FUNCTION F_ITC_SendRTR : BOOL
(**************************************************************************************
 * 	Application		:	BoxControl Framework
 *	Revision		:	$Revision: 404529 $
 *	Revision date	:	$Date: 2018-04-23 08:21:38 +0200 (Mo., 23 Apr 2018) $
 *	Last changed by	:	$Author: b7bolm $
 *	URL				:	$URL: http://almscdc.swisslog.com/repo/SWPD/Development/BoxControlFramework/20_Release/trunk/01_Software/BCF/BCF/JumpStart/20_Product/10_App/11_Com/10_Lib/10_Conv/11_ITC/F_ITC_SendRTR.TcPOU $
 *
 *	Purpose			:	Wrap message - RTR
 *
 * ------------------------------------------------------------------------------------
 *	Copyright Swisslog [IP AG], Switzerland. All rights reserved.
 * 
 * ------------------------------------------------------------------------------------
 *	
 * 	Revision History: 
 *
 * 	VERSION			DATE			INITIALS			DESCRIPTION
 *	0.1				01.01.2001		swl					Example
 *
 **************************************************************************************)
VAR_INPUT
	eChannelSrc		: E_MFCS_Channel; // Source communicaton channel
	PositionName	: STRING(Conveyor.POSITION_STRINGLENGTH); // SIS MM-GGG-EEEE-FF-Z
	eReturnCode		: E_ErrorConv; // Return code
END_VAR
VAR
	RTR				: ST_ITC_RTR; 
END_VAR

// Map values
RTR.Position := PositionName;
RTR.ReturnCode := eReturnCode;

// Forward to ITC
F_ITC_SendRTR := fbITC_Manager.M_SendData(
					meChannel	:= eChannelSrc,
					mMsgType	:= E_ITC_MsgTypeConv.E_REMOVE_TU_REPORT,
					mpData		:= ADR(RTR),
					mLen		:= SIZEOF(RTR));

END_FUNCTION

(* stored: Version 1.1.0.1, ProductVersion 3.1.4022.12
   POU F_ITC_SendRTR: Id {80b2f679-8988-42f8-a8ea-efc42201546f}, SpecialFunc None *)
